PROGRAM Stop
VAR
	Stop_Button:BOOL;
	Break_At_Home: BOOL;
END_VAR

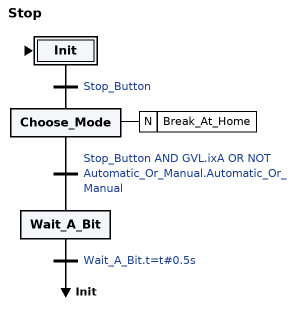
INITIAL_STEP Init:
END_STEP
TRANSITION FROM Init TO Choose_Mode
    := Stop_Button;
END_TRANSITION
STEP Choose_Mode:
    Break_At_Home(N);
END_STEP
TRANSITION FROM Choose_Mode TO Wait_A_Bit
    := Stop_Button AND GVL.ixA OR NOT Automatic_Or_Manual.Automatic_Or_Manual;
END_TRANSITION
STEP Wait_A_Bit:
END_STEP
TRANSITION FROM Wait_A_Bit TO Init
    := Wait_A_Bit.t=t#0.5s;
END_TRANSITION

END_PROGRAM

(* stored: Version 1.1.0.1, ProductVersion 3.1.4024.12
   POU Stop: Id {35ca82df-c971-4e35-b3a4-b60f9d096624}, SpecialFunc None *)
